FUNCTION F_DrawOrientation : HRESULT
VAR_INPUT
    ipSrcImage  : ITcVnImage;
    ipDestImage : Reference To  ITcVnImage;
    eTransform  : ETcVnColorSpaceTransform;
    hrPrev      : HRESULT;
END_VAR
VAR
	ipContourList	: ITcVnContainer;
	ipIterator		: ITcVnForwardIterator;
	ipContour		: ITcVnContainer;
	
	fArea                 :    LREAL;
	fAreaMin              :    LREAL := 100;
	fAreaMax              :    LREAL := 100000;
END_VAR

hrPrev := F_VN_FindContours(ipSrcImage,ipContourList,hrPrev);
hrPrev := F_VN_GetForwardIterator(ipContourList, ipIterator, hrPrev);

WHILE SUCCEEDED(hrPrev) AND_THEN ipIterator.CheckIfEnd() <> S_OK DO
	hrPrev := F_VN_GetContainer(ipIterator, ipContour,hrPrev);
	hrPrev := F_VN_IncrementIterator(ipIterator,hrPrev);
	
	// Filter by Area
    hrPrev := F_VN_ContourArea(ipContour, fArea, hrPrev);
	
	IF fArea > fAreaMin AND fArea < fAreaMax THEN
		hrPrev := F_GetOrientationST(
	END_IF
END_WHILE

END_FUNCTION

(* stored: Version 1.1.0.1, ProductVersion 3.1.4024.12
   POU F_DrawOrientation: Id {bd828471-7398-4d25-a4e8-8b31d8284100}, SpecialFunc None *)
